INTERFACE I_LinkedListDisposedEvent EXTENDS I_Event

PROPERTY PUBLIC TargetLinkedList : I_LinkedList
GET
END_GET
END_PROPERTY

END_INTERFACE

(* stored: Version 1.1.0.1, ProductVersion 3.1.4024.12
   Itf I_LinkedListDisposedEvent: Id {28133386-e3b6-4050-8ebb-01e97c0da9dd}
   Property TargetLinkedList: Id {d9c40f2b-abbd-40ff-872b-dd59aad32e4c}
   Get Get: Id {1329a907-adfd-4d2c-ad5a-a0f4a118da38} *)
